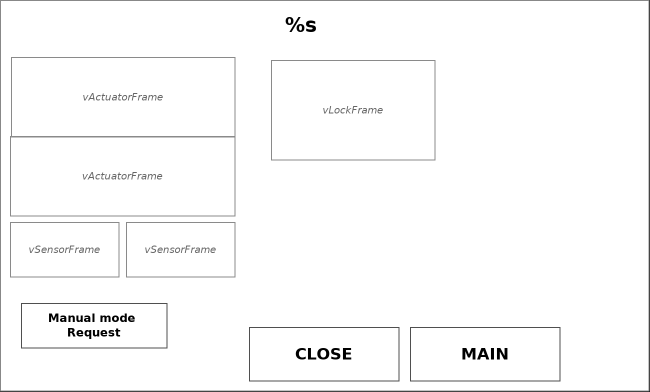
VISUALIZATION vTableWeighingService  // 650x392
VAR_IN_OUT
	fbStation:FB_WeighingStation;
	fbTableControl: FB_TableControl;
END_VAR
    Rectangle (0,0 650x392)
    Rectangle (21,303 146x45), "Manual mode Request", colour toggle: fbStation.bManualModeActive
        toggle fbStation.bManualModeRequest
    Rectangle (226,10 150x30), "%s", text variable: fbStation.sStationName
    Frame (10,136 225x80)
        shows vActuatorFrame(iTextIndex1 := 0, iTextIndex2 := 1, fbActuator := fbStation.fbWeighingActuator)
    Frame (11,57 224x80)
        shows vActuatorFrame(iTextIndex1 := 2, iTextIndex2 := 3, fbActuator := fbStation.fbPusherActuator)
    Frame (10,222 109x55)
        shows vSensorFrame(iNameIndex := 1, fbSensor := fbStation.fbBottleSensor)
    Frame (126,222 109x55)
        shows vSensorFrame(iNameIndex := 2, fbSensor := fbStation.fbBottleDrawerSensor)
    Frame (271,60 164x100)
        shows vLockFrame(iNameIndex := 3, fbLock := fbStation.fbDrawerLock)
    Rectangle (410,327 150x54), "MAIN"
        OnMouseDown: execute { fbTableControl.stHMI.iDialogNumber:=201; }
    Rectangle (249,327 150x54), "CLOSE"
        OnMouseDown: execute { fbTableControl.stHMI.iDialogNumber:=0; }
END_VISUALIZATION

(* stored: Version 1.1.0.1, ProductVersion 3.1.4024.15
   Visu vTableWeighingService: Id {3fb1c437-625a-4e18-a9dd-bdc0feac539c} *)
